FUNCTION Convert_USINT_TO_DINT : Hresult
VAR_INPUT
	in : USINT;
	out : REFERENCE TO DINT;
END_VAR
VAR
	converted : DINT;
END_VAR

converted := USINT_TO_DINT(in);

IF (DINT_TO_USINT(converted) <> in) THEN
	Convert_USINT_TO_DINT := INCOMPATIBLE;
	RETURN;
END_IF

out := converted;

END_FUNCTION

(* stored: Version 1.1.0.1, ProductVersion 3.1.4024.12
   POU Convert_USINT_TO_DINT: Id {f6e2687e-0e0b-408a-aec8-c960e8ff1563}, SpecialFunc None *)
